	X =  321.485  mm,	Y =   -468.955  mm,	Z =   -267.000  mm,
	W =  90.000 deg,	P =   0.000 deg,	R =   90.000 deg
};
P[439]{
   GP1:
	UF : 0, UT : 6,		CONFIG : 'N U T, 0, 0, 0',
	X =  303.278  mm,	Y =   -479.431  mm,	Z =   -267.000  mm,
	W =  90.000 deg,	P =   0.000 deg,	R =   90.000 deg
};
P[440]{
   GP1:
	UF : 0, UT : 6,		CONFIG : 'N U T, 0, 0, 0',
	X =  248.887  mm,	Y =   -510.794  mm,	Z =   -267.000  mm,
	W =  90.000 deg,	P =   0.000 deg,	R =   90.000 deg
};
P[441]{
   GP1:
	UF : 0, UT : 6,		CONFIG : 'N U T, 0, 0, 0',
	X =  230.541  mm,	Y =   -521.505  mm,	Z =   -267.000  mm,
	W =  90.000 deg,	P =   0.000 deg,	R =   90.000 deg
};
P[442]{
   GP1:
	UF : 0, UT : 6,		CONFIG : 'N U T, 0, 0, 0',
	X =  194.065  mm,	Y =   -542.556  mm,	Z =   -267.000  mm,
	W =  90.000 deg,	P =   0.000 deg,	R =   90.000 deg
};
P[443]{
   GP1:
	UF : 0, UT : 6,		CONFIG : 'N U T, 0, 0, 0',
	X =  139.530  mm,	Y =   -573.935  mm,	Z =   -267.000  mm,
	W =  90.000 deg,	P =   0.000 deg,	R =   90.000 deg
};
P[444]{
   GP1:
	UF : 0, UT : 6,		CONFIG : 'N U T, 0, 0, 0',
	X =  121.558  mm,	Y =   -584.313  mm,	Z =   -267.000  mm,
	W =  90.000 deg,	P =   0.000 deg,	R =   90.000 deg
};
P[445]{
   GP1:
	UF : 0, UT : 6,		CONFIG : 'N U T, 0, 0, 0',
	X =  69.455  mm,	Y =   -614.511  mm,	Z =   -248.193  mm,
	W =  90.000 deg,	P =   0.000 deg,	R =   90.000 deg
};
P[446]{
   GP1:
	UF : 0, UT : 6,		CONFIG : 'N U T, 0, 0, 0',
	X =  73.807  mm,	Y =   -612.144  mm,	Z =   -261.927  mm,
	W =  90.000 deg,	P =   0.000 deg,	R =   90.000 deg
};
P[447]{
   GP1:
	UF : 0, UT : 6,		CONFIG : 'N U T, 0, 0, 0',
	X =  85.175  mm,	Y =   -605.574  mm,	Z =   -266.999  mm,
	W =  90.000 deg,	P =   0.000 deg,	R =   90.000 deg
};
P[448]{
   GP1:
	UF : 0, UT : 6,		CONFIG : 'N U T, 0, 0, 0',
	X =  103.342  mm,	Y =   -595.091  mm,	Z =   -267.000  mm,
	W =  90.000 deg,	P =   0.000 deg,	R =   90.000 deg
};
P[449]{
   GP1:
	UF : 0, UT : 6,		CONFIG : 'N U T, 0, 0, 0',
	X =  158.046  mm,	Y =   -563.598  mm,	Z =   -267.000  mm,
	W =  90.000 deg,	P =   0.000 deg,	R =   90.000 deg
};
P[450]{
   GP1:
	UF : 0, UT : 6,		CONFIG : 'N U T, 0, 0, 0',
	X =  176.088  mm,	Y =   -553.101  mm,	Z =   -267.000  mm,
	W =  90.000 deg,	P =   0.000 deg,	R =   90.000 deg
};
P[451]{
   GP1:
	UF : 0, UT : 6,		CONFIG : 'N U T, 0, 0, 0',
	X =  212.495  mm,	Y =   -531.950  mm,	Z =   -267.000  mm,
	W =  90.000 deg,	P =   0.000 deg,	R =   90.000 deg
};
P[452]{
   GP1:
	UF : 0, UT : 6,		CONFIG : 'N U T, 0, 0, 0',
	X =  266.860  mm,	Y =   -500.614  mm,	Z =   -267.000  mm,
	W =  90.000 deg,	P =   0.000 deg,	R =   90.000 deg
};
P[453]{
   GP1:
	UF : 0, UT : 6,		CONFIG : 'N U T, 0, 0, 0',
	X =  285.368  mm,	Y =   -490.006  mm,	Z =   -267.000  mm,
	W =  90.000 deg,	P =   0.000 deg,	R =   90.000 deg
};
P[454]{
   GP1:
	UF : 0, UT : 6,		CONFIG : 'N U T, 0, 0, 0',
	X =  339.837  mm,	Y =   -458.448  mm,	Z =   -267.000  mm,
	W =  90.000 deg,	P =   0.000 deg,	R =   90.000 deg
};
P[455]{
   GP1:
	UF : 0, UT : 6,		CONFIG : 'N U T, 0, 0, 0',
	X =  357.990  mm,	Y =   -448.207  mm,	Z =   -267.000  mm,
	W =  90.000 deg,	P =   0.000 deg,	R =   90.000 deg
};
P[456]{
   GP1:
	UF : 0, UT : 6,		CONFIG : 'N U T, 0, 0, 0',
	X =  376.120  mm,	Y =   -437.531  mm,	Z =   -267.000  mm,
	W =  90.000 deg,	P =   0.000 deg,	R =   90.000 deg
};
P[457]{
   GP1:
	UF : 0, UT : 6,		CONFIG : 'N U T, 0, 0, 0',
	X =  394.238  mm,	Y =   -427.152  mm,	Z =   -267.000  mm,
	W =  90.000 deg,	P =   0.000 deg,	R =   90.000 deg
};
P[458]{
   GP1:
	UF : 0, UT : 6,		CONFIG : 'N U T, 0, 0, 0',
	X =  412.785  mm,	Y =   -416.547  mm,	Z =   -267.000  mm,
	W =  90.000 deg,	P =   0.000 deg,	R =   90.000 deg
};
P[459]{
   GP1:
	UF : 0, UT : 6,		CONFIG : 'N U T, 0, 0, 0',
	X =  448.959  mm,	Y =   -395.706  mm,	Z =   -267.000  mm,
	W =  90.000 deg,	P =   0.000 deg,	R =   90.000 deg
};
P[460]{
   GP1:
	UF : 0, UT : 6,		CONFIG : 'N U T, 0, 0, 0',
	X =  485.175  mm,	Y =   -374.654  mm,	Z =   -267.000  mm,
	W =  90.000 deg,	P =   0.000 deg,	R =   90.000 deg
};
P[461]{
   GP1:
	UF : 0, UT : 6,		CONFIG : 'N U T, 0, 0, 0',
	X =  521.461  mm,	Y =   -353.543  mm,	Z =   -267.000  mm,
	W =  90.000 deg,	P =   0.000 deg,	R =   90.000 deg
};
P[462]{
   GP1:
	UF : 0, UT : 6,		CONFIG : 'N U T, 0, 0, 0',
	X =  581.548  mm,	Y =   -343.057  mm,	Z =   -248.136  mm,
	W =  90.000 deg,	P =   0.000 deg,	R =   90.000 deg
};
P[463]{
   GP1:
	UF : 0, UT : 6,		CONFIG : 'N U T, 0, 0, 0',
	X =  569.674  mm,	Y =   -349.887  mm,	Z =   -266.231  mm,
	W =  90.000 deg,	P =   0.000 deg,	R =   90.000 deg
};
P[464]{
   GP1:
	UF : 0, UT : 6,		CONFIG : 'N U T, 0, 0, 0',
	X =  495.732  mm,	Y =   -392.513  mm,	Z =   -267.000  mm,
	W =  90.000 deg,	P =   0.000 deg,	R =   90.000 deg
};
P[465]{
   GP1:
	UF : 0, UT : 6,		CONFIG : 'N U T, 0, 0, 0',
	X =  477.461  mm,	Y =   -403.017  mm,	Z =   -267.000  mm,
	W =  90.000 deg,	P =   0.000 deg,	R =   90.000 deg
};
P[466]{
   GP1:
	UF : 0, UT : 6,		CONFIG : 'N U T, 0, 0, 0',
	X =  441.221  mm,	Y =   -424.060  mm,	Z =   -267.000  mm,
	W =  90.000 deg,	P =   0.000 deg,	R =   90.000 deg
};
P[467]{
   GP1:
	UF : 0, UT : 6,		CONFIG : 'N U T, 0, 0, 0',
	X =  404.597  mm,	Y =   -445.232  mm,	Z =   -267.000  mm,
	W =  90.000 deg,	P =   0.000 deg,	R =   90.000 deg
};
P[468]{
   GP1:
	UF : 0, UT : 6,		CONFIG : 'N U T, 0, 0, 0',
	X =  386.626  mm,	Y =   -455.612  mm,	Z =   -267.000  mm,
	W =  90.000 deg,	P =   0.000 deg,	R =   90.000 deg
};
P[469]{
   GP1:
	UF : 0, UT : 6,		CONFIG : 'N U T, 0, 0, 0',
	X =  368.349  mm,	Y =   -466.118  mm,	Z =   -267.000  mm,
	W =  90.000 deg,	P =   0.000 deg,	R =   90.000 deg
};
P[470]{
   GP1:
	UF : 0, UT : 6,		CONFIG : 'N U T, 0, 0, 0',
	X =  350.098  mm,	Y =   -476.669  mm,	Z =   -267.000  mm,
	W =  90.000 deg,	P =   0.000 deg,	R =   90.000 deg
};
P[471]{
   GP1:
	UF : 0, UT : 6,		CONFIG : 'N U T, 0, 0, 0',
	X =  313.809  mm,	Y =   -497.611  mm,	Z =   -267.000  mm,
	W =  90.000 deg,	P =   0.000 deg,	R =   90.000 deg
};
P[472]{
   GP1:
	UF : 0, UT : 6,		CONFIG : 'N U T, 0, 0, 0',
	X =  259.253  mm,	Y =   -529.033  mm,	Z =   -267.000  mm,
	W =  90.000 deg,	P =   0.000 deg,	R =   90.000 deg
};
P[473]{
   GP1:
	UF : 0, UT : 6,		CONFIG : 'N U T, 0, 0, 0',
	X =  240.975  mm,	Y =   -539.441  mm,	Z =   -267.000  mm,
	W =  90.000 deg,	P =   0.000 deg,	R =   90.000 deg
};
P[474]{
   GP1:
	UF : 0, UT : 6,		CONFIG : 'N U T, 0, 0, 0',
	X =  186.337  mm,	Y =   -571.044  mm,	Z =   -267.000  mm,
	W =  90.000 deg,	P =   0.000 deg,	R =   90.000 deg
};
P[475]{
   GP1:
	UF : 0, UT : 6,		CONFIG : 'N U T, 0, 0, 0',
	X =  131.747  mm,	Y =   -602.648  mm,	Z =   -267.000  mm,
	W =  90.000 deg,	P =   0.000 deg,	R =   90.000 deg
};
P[476]{
   GP1:
	UF : 0, UT : 6,		CONFIG : 'N U T, 0, 0, 0',
	X =  113.540  mm,	Y =   -613.030  mm,	Z =   -267.000  mm,
	W =  90.000 deg,	P =   0.000 deg,	R =   90.000 deg
};
P[477]{
   GP1:
	UF : 0, UT : 6,		CONFIG : 'N U T, 0, 0, 0',
	X =  79.956  mm,	Y =   -632.694  mm,	Z =   -248.200  mm,
	W =  90.000 deg,	P =   0.000 deg,	R =   90.000 deg
};
P[478]{
   GP1:
	UF : 0, UT : 6,		CONFIG : 'N U T, 0, 0, 0',
	X =  84.360  mm,	Y =   -630.389  mm,	Z =   -261.973  mm,
	W =  90.000 deg,	P =   0.000 deg,	R =   90.000 deg
};
P[479]{
   GP1:
	UF : 0, UT : 6,		CONFIG : 'N U T, 0, 0, 0',
	X =  95.519  mm,	Y =   -623.823  mm,	Z =   -266.999  mm,
	W =  90.000 deg,	P =   0.000 deg,	R =   90.000 deg
};
P[480]{
   GP1:
	UF : 0, UT : 6,		CONFIG : 'N U T, 0, 0, 0',
	X =  150.126  mm,	Y =   -592.253  mm,	Z =   -267.000  mm,
	W =  90.000 deg,	P =   0.000 deg,	R =   90.000 deg
};
P[481]{
   GP1:
	UF : 0, UT : 6,		CONFIG : 'N U T, 0, 0, 0',
	X =  168.419  mm,	Y =   -581.719  mm,	Z =   -267.000  mm,
	W =  90.000 deg,	P =   0.000 deg,	R =   90.000 deg
};
P[482]{
   GP1:
	UF : 0, UT : 6,		CONFIG : 'N U T, 0, 0, 0',
	X =  204.831  mm,	Y =   -560.612  mm,	Z =   -267.000  mm,
	W =  90.000 deg,	P =   0.000 deg,	R =   90.000 deg
};
P[483]{
   GP1:
	UF : 0, UT : 6,		CONFIG : 'N U T, 0, 0, 0',
	X =  223.052  mm,	Y =   -550.261  mm,	Z =   -267.000  mm,
	W =  90.000 deg,	P =   0.000 deg,	R =   90.000 deg
};
P[484]{
   GP1:
	UF : 0, UT : 6,		CONFIG : 'N U T, 0, 0, 0',
	X =  277.625  mm,	Y =   -518.677  mm,	Z =   -267.000  mm,
	W =  90.000 deg,	P =   0.000 deg,	R =   90.000 deg
};
P[485]{
   GP1:
	UF : 0, UT : 6,		CONFIG : 'N U T, 0, 0, 0',
	X =  295.801  mm,	Y =   -508.256  mm,	Z =   -267.000  mm,
	W =  90.000 deg,	P =   0.000 deg,	R =   90.000 deg
};
P[486]{
   GP1:
	UF : 0, UT : 6,		CONFIG : 'N U T, 0, 0, 0',
	X =  332.180  mm,	Y =   -487.237  mm,	Z =   -267.000  mm,
	W =  90.000 deg,	P =   0.000 deg,	R =   90.000 deg
};
P[487]{
   GP1:
	UF : 0, UT : 6,		CONFIG : 'N U T, 0, 0, 0',
	X =  422.842  mm,	Y =   -434.745  mm,	Z =   -267.000  mm,
	W =  90.000 deg,	P =   0.000 deg,	R =   90.000 deg
};
P[488]{
   GP1:
	UF : 0, UT : 6,		CONFIG : 'N U T, 0, 0, 0',
	X =  459.065  mm,	Y =   -413.887  mm,	Z =   -267.000  mm,
	W =  90.000 deg,	P =   0.000 deg,	R =   90.000 deg
};
P[489]{
   GP1:
	UF : 0, UT : 6,		CONFIG : 'N U T, 0, 0, 0',
	X =  514.184  mm,	Y =   -382.024  mm,	Z =   -267.000  mm,
	W =  90.000 deg,	P =   0.000 deg,	R =   90.000 deg
};
P[490]{
   GP1:
	UF : 0, UT : 6,		CONFIG : 'N U T, 0, 0, 0',
	X =  532.228  mm,	Y =   -371.647  mm,	Z =   -267.000  mm,
	W =  90.000 deg,	P =   0.000 deg,	R =   90.000 deg
};
P[491]{
   GP1:
	UF : 0, UT : 6,		CONFIG : 'N U T, 0, 0, 0',
	X =  550.141  mm,	Y =   -361.240  mm,	Z =   -267.000  mm,
	W =  90.000 deg,	P =   0.000 deg,	R =   90.000 deg
};
P[492]{
   GP1:
	UF : 0, UT : 6,		CONFIG : 'N U T, 0, 0, 0',
	X =  578.422  mm,	Y =   -345.240  mm,	Z =   -258.781  mm,
	W =  90.000 deg,	P =   0.000 deg,	R =   90.000 deg
};
P[493]{
   GP1:
	UF : 0, UT : 6,		CONFIG : 'N U T, 0, 0, 0',
	X =  580.211  mm,	Y =   -368.067  mm,	Z =   -266.283  mm,
	W =  90.000 deg,	P =   0.000 deg,	R =   90.000 deg
};
P[494]{
   GP1:
	UF : 0, UT : 6,		CONFIG : 'N U T, 0, 0, 0',
	X =  560.695  mm,	Y =   -379.290  mm,	Z =   -267.000  mm,
	W =  90.000 deg,	P =   0.000 deg,	R =   90.000 deg
};
P[495]{
   GP1:
	UF : 0, UT : 6,		CONFIG : 'N U T, 0, 0, 0',
	X =  505.985  mm,	Y =   -410.945  mm,	Z =   -267.000  mm,
	W =  90.000 deg,	P =   0.000 deg,	R =   90.000 deg
};
P[496]{
   GP1:
	UF : 0, UT : 6,		CONFIG : 'N U T, 0, 0, 0',
	X =  469.806  mm,	Y =   -431.829  mm,	Z =   -267.000  mm,
	W =  90.000 deg,	P =   0.000 deg,	R =   90.000 deg
};
P[497]{
   GP1:
	UF : 0, UT : 6,		CONFIG : 'N U T, 0, 0, 0',
	X =  396.987  mm,	Y =   -473.854  mm,	Z =   -267.000  mm,
	W =  90.000 deg,	P =   0.000 deg,	R =   90.000 deg
};
P[498]{
   GP1:
	UF : 0, UT : 6,		CONFIG : 'N U T, 0, 0, 0',
	X =  360.530  mm,	Y =   -494.814  mm,	Z =   -267.000  mm,
	W =  90.000 deg,	P =   0.000 deg,	R =   90.000 deg
};
P[499]{
   GP1:
	UF : 0, UT : 6,		CONFIG : 'N U T, 0, 0, 0',
	X =  342.478  mm,	Y =   -505.311  mm,	Z =   -267.000  mm,
	W =  90.000 deg,	P =   0.000 deg,	R =   90.000 deg
};
P[500]{
   GP1:
	UF : 0, UT : 6,		CONFIG : 'N U T, 0, 0, 0',
	X =  324.052  mm,	Y =   -515.696  mm,	Z =   -267.000  mm,
	W =  90.000 deg,	P =   0.000 deg,	R =   90.000 deg
};
P[501]{
   GP1:
	UF : 0, UT : 6,		CONFIG : 'N U T, 0, 0, 0',
	X =  306.123  mm,	Y =   -526.319  mm,	Z =   -267.000  mm,
	W =  90.000 deg,	P =   0.000 deg,	R =   90.000 deg
};
P[502]{
   GP1:
	UF : 0, UT : 6,		CONFIG : 'N U T, 0, 0, 0',
	X =  287.949  mm,	Y =   -536.712  mm,	Z =   -267.000  mm,
	W =  90.000 deg,	P =   0.000 deg,	R =   90.000 deg
};
P[503]{
   GP1:
	UF : 0, UT : 6,		CONFIG : 'N U T, 0, 0, 0',
	X =  251.698  mm,	Y =   -557.782  mm,	Z =   -267.000  mm,
	W =  90.000 deg,	P =   0.000 deg,	R =   90.000 deg
};
P[504]{
   GP1:
	UF : 0, UT : 6,		CONFIG : 'N U T, 0, 0, 0',
	X =  215.213  mm,	Y =   -578.773  mm,	Z =   -267.000  mm,
	W =  90.000 deg,	P =   0.000 deg,	R =   90.000 deg
};
P[505]{
   GP1:
	UF : 0, UT : 6,		CONFIG : 'N U T, 0, 0, 0',
	X =  160.535  mm,	Y =   -610.339  mm,	Z =   -267.000  mm,
	W =  90.000 deg,	P =   0.000 deg,	R =   90.000 deg
};
P[506]{
   GP1:
	UF : 0, UT : 6,		CONFIG : 'N U T, 0, 0, 0',
	X =  142.213  mm,	Y =   -620.805  mm,	Z =   -267.000  mm,
	W =  90.000 deg,	P =   0.000 deg,	R =   90.000 deg
};
P[507]{
   GP1:
	UF : 0, UT : 6,		CONFIG : 'N U T, 0, 0, 0',
	X =  106.162  mm,	Y =   -641.800  mm,	Z =   -266.999  mm,
	W =  90.000 deg,	P =   0.000 deg,	R =   90.000 deg
};
P[508]{
   GP1:
	UF : 0, UT : 6,		CONFIG : 'N U T, 0, 0, 0',
	X =  94.773  mm,	Y =   -648.395  mm,	Z =   -262.002  mm,
	W =  90.000 deg,	P =   0.000 deg,	R =   90.000 deg
};
P[509]{
   GP1:
	UF : 0, UT : 6,		CONFIG : 'N U T, 0, 0, 0',
	X =  90.472  mm,	Y =   -650.908  mm,	Z =   -248.200  mm,
	W =  90.000 deg,	P =   0.000 deg,	R =   90.000 deg
};
P[510]{
   GP1:
	UF : 0, UT : 6,		CONFIG : 'N U T, 0, 0, 0',
	X =  124.271  mm,	Y =   -631.447  mm,	Z =   -267.000  mm,
	W =  90.000 deg,	P =   0.000 deg,	R =   90.000 deg
};
P[511]{
   GP1:
	UF : 0, UT : 6,		CONFIG : 'N U T, 0, 0, 0',
	X =  178.773  mm,	Y =   -600.003  mm,	Z =   -267.000  mm,
	W =  90.000 deg,	P =   0.000 deg,	R =   90.000 deg
};
P[512]{
   GP1:
	UF : 0, UT : 6,		CONFIG : 'N U T, 0, 0, 0',
	X =  196.986  mm,	Y =   -589.631  mm,	Z =   -267.000  mm,
	W =  90.000 deg,	P =   0.000 deg,	R =   90.000 deg
};
P[513]{
   GP1:
	UF : 0, UT : 6,		CONFIG : 'N U T, 0, 0, 0',
	X =  233.418  mm,	Y =   -568.352  mm,	Z =   -267.000  mm,
	W =  90.000 deg,	P =   0.000 deg,	R =   90.000 deg
};
P[514]{
   GP1:
	UF : 0, UT : 6,		CONFIG : 'N U T, 0, 0, 0',
	X =  269.919  mm,	Y =   -547.346  mm,	Z =   -267.000  mm,
	W =  90.000 deg,	P =   0.000 deg,	R =   90.000 deg
};
P[515]{
   GP1:
	UF : 0, UT : 6,		CONFIG : 'N U T, 0, 0, 0',
	X =  378.875  mm,	Y =   -484.547  mm,	Z =   -267.000  mm,
	W =  90.000 deg,	P =   0.000 deg,	R =   90.000 deg
};
P[516]{
   GP1:
	UF : 0, UT : 6,		CONFIG : 'N U T, 0, 0, 0',
	X =  415.424  mm,	Y =   -463.320  mm,	Z =   -267.000  mm,
	W =  90.000 deg,	P =   0.000 deg,	R =   90.000 deg
};
P[517]{
   GP1:
	UF : 0, UT : 6,		CONFIG : 'N U T, 0, 0, 0',
	X =  433.559  mm,	Y =   -452.991  mm,	Z =   -267.000  mm,
	W =  90.000 deg,	P =   0.000 deg,	R =   90.000 deg
};
P[518]{
   GP1:
	UF : 0, UT : 6,		CONFIG : 'N U T, 0, 0, 0',
	X =  451.784  mm,	Y =   -442.412  mm,	Z =   -267.000  mm,
	W =  90.000 deg,	P =   0.000 deg,	R =   90.000 deg
};
P[519]{
   GP1:
	UF : 0, UT : 6,		CONFIG : 'N U T, 0, 0, 0',
	X =  488.126  mm,	Y =   -421.292  mm,	Z =   -267.000  mm,
	W =  90.000 deg,	P =   0.000 deg,	R =   90.000 deg
};
P[520]{
   GP1:
	UF : 0, UT : 6,		CONFIG : 'N U T, 0, 0, 0',
	X =  524.439  mm,	Y =   -400.389  mm,	Z =   -267.000  mm,
	W =  90.000 deg,	P =   0.000 deg,	R =   90.000 deg
};
P[521]{
   GP1:
	UF : 0, UT : 6,		CONFIG : 'N U T, 0, 0, 0',
	X =  542.644  mm,	Y =   -390.001  mm,	Z =   -267.000  mm,
	W =  90.000 deg,	P =   0.000 deg,	R =   90.000 deg
};
P[522]{
   GP1:
	UF : 0, UT : 6,		CONFIG : 'N U T, 0, 0, 0',
	X =  588.832  mm,	Y =   -363.325  mm,	Z =   -258.859  mm,
	W =  90.000 deg,	P =   0.000 deg,	R =   90.000 deg
};
P[523]{
   GP1:
	UF : 0, UT : 6,		CONFIG : 'N U T, 0, 0, 0',
	X =  592.208  mm,	Y =   -361.394  mm,	Z =   -247.960  mm,
	W =  90.000 deg,	P =   0.000 deg,	R =   90.000 deg
};
P[524]{
   GP1:
	UF : 0, UT : 6,		CONFIG : 'N U T, 0, 0, 0',
	X =  602.472  mm,	Y =   -379.509  mm,	Z =   -248.435  mm,
	W =  90.000 deg,	P =   0.000 deg,	R =   90.000 deg
};
P[525]{
   GP1:
	UF : 0, UT : 6,		CONFIG : 'N U T, 0, 0, 0',
	X =  534.847  mm,	Y =   -418.347  mm,	Z =   -267.000  mm,
	W =  90.000 deg,	P =   0.000 deg,	R =   90.000 deg
};
P[526]{
   GP1:
	UF : 0, UT : 6,		CONFIG : 'N U T, 0, 0, 0',
	X =  498.274  mm,	Y =   -439.482  mm,	Z =   -267.000  mm,
	W =  90.000 deg,	P =   0.000 deg,	R =   90.000 deg
};
P[527]{
   GP1:
	UF : 0, UT : 6,		CONFIG : 'N U T, 0, 0, 0',
	X =  407.652  mm,	Y =   -491.986  mm,	Z =   -267.000  mm,
	W =  90.000 deg,	P =   0.000 deg,	R =   90.000 deg
};
P[528]{
   GP1:
	UF : 0, UT : 6,		CONFIG : 'N U T, 0, 0, 0',
	X =  389.393  mm,	Y =   -502.496  mm,	Z =   -267.000  mm,
	W =  90.000 deg,	P =   0.000 deg,	R =   90.000 deg
};
P[529]{
   GP1:
	UF : 0, UT : 6,		CONFIG : 'N U T, 0, 0, 0',
	X =  352.833  mm,	Y =   -523.469  mm,	Z =   -267.000  mm,
	W =  90.000 deg,	P =   0.000 deg,	R =   90.000 deg
};
P[530]{
   GP1:
	UF : 0, UT : 6,		CONFIG : 'N U T, 0, 0, 0',
	X =  316.604  mm,	Y =   -544.429  mm,	Z =   -267.000  mm,
	W =  90.000 deg,	P =   0.000 deg,	R =   90.000 deg
};
P[531]{
   GP1:
	UF : 0, UT : 6,		CONFIG : 'N U T, 0, 0, 0',
	X =  280.341  mm,	Y =   -565.474  mm,	Z =   -267.000  mm,
	W =  90.000 deg,	P =   0.000 deg,	R =   90.000 deg
};
P[532]{
   GP1:
	UF : 0, UT : 6,		CONFIG : 'N U T, 0, 0, 0',
	X =  243.658  mm,	Y =   -586.484  mm,	Z =   -267.000  mm,
	W =  90.000 deg,	P =   0.000 deg,	R =   90.000 deg
};
P[533]{
   GP1:
	UF : 0, UT : 6,		CONFIG : 'N U T, 0, 0, 0',
	X =  225.600  mm,	Y =   -596.805  mm,	Z =   -267.000  mm,
	W =  90.000 deg,	P =   0.000 deg,	R =   90.000 deg
};
P[534]{
   GP1:
	UF : 0, UT : 6,		CONFIG : 'N U T, 0, 0, 0',
	X =  207.565  mm,	Y =   -607.525  mm,	Z =   -267.000  mm,
	W =  90.000 deg,	P =   0.000 deg,	R =   90.000 deg
};
P[535]{
   GP1:
	UF : 0, UT : 6,		CONFIG : 'N U T, 0, 0, 0',
	X =  134.641  mm,	Y =   -649.517  mm,	Z =   -267.000  mm,
	W =  90.000 deg,	P =   0.000 deg,	R =   90.000 deg
};
P[536]{
   GP1:
	UF : 0, UT : 6,		CONFIG : 'N U T, 0, 0, 0',
	X =  116.667  mm,	Y =   -659.834  mm,	Z =   -266.999  mm,
	W =  90.000 deg,	P =   0.000 deg,	R =   90.000 deg
};
P[537]{
   GP1:
	UF : 0, UT : 6,		CONFIG : 'N U T, 0, 0, 0',
	X =  100.943  mm,	Y =   -669.018  mm,	Z =   -248.233  mm,
	W =  90.000 deg,	P =   0.000 deg,	R =   90.000 deg
};
P[538]{
   GP1:
	UF : 0, UT : 6,		CONFIG : 'N U T, 0, 0, 0',
	X =  105.313  mm,	Y =   -666.641  mm,	Z =   -261.991  mm,
	W =  90.000 deg,	P =   0.000 deg,	R =   90.000 deg
};
P[539]{
   GP1:
	UF : 0, UT : 6,		CONFIG : 'N U T, 0, 0, 0',
	X =  152.979  mm,	Y =   -639.046  mm,	Z =   -267.000  mm,
	W =  90.000 deg,	P =   0.000 deg,	R =   90.000 deg
};
P[540]{
   GP1:
	UF : 0, UT : 6,		CONFIG : 'N U T, 0, 0, 0',
	X =  171.400  mm,	Y =   -628.527  mm,	Z =   -267.000  mm,
	W =  90.000 deg,	P =   0.000 deg,	R =   90.000 deg
};
P[541]{
   GP1:
	UF : 0, UT : 6,		CONFIG : 'N U T, 0, 0, 0',
	X =  189.254  mm,	Y =   -618.287  mm,	Z =   -267.000  mm,
	W =  90.000 deg,	P =   0.000 deg,	R =   90.000 deg
};
P[542]{
   GP1:
	UF : 0, UT : 6,		CONFIG : 'N U T, 0, 0, 0',
	X =  261.985  mm,	Y =   -576.181  mm,	Z =   -267.000  mm,
	W =  90.000 deg,	P =   0.000 deg,	R =   90.000 deg
};
P[543]{
   GP1:
	UF : 0, UT : 6,		CONFIG : 'N U T, 0, 0, 0',
	X =  298.625  mm,	Y =   -555.072  mm,	Z =   -267.000  mm,
	W =  90.000 deg,	P =   0.000 deg,	R =   90.000 deg
};
P[544]{
   GP1:
	UF : 0, UT : 6,		CONFIG : 'N U T, 0, 0, 0',
	X =  334.764  mm,	Y =   -534.219  mm,	Z =   -267.000  mm,
	W =  90.000 deg,	P =   0.000 deg,	R =   90.000 deg
};
P[545]{
   GP1:
	UF : 0, UT : 6,		CONFIG : 'N U T, 0, 0, 0',
	X =  371.261  mm,	Y =   -513.223  mm,	Z =   -267.000  mm,
	W =  90.000 deg,	P =   0.000 deg,	R =   90.000 deg
};
P[546]{
   GP1:
	UF : 0, UT : 6,		CONFIG : 'N U T, 0, 0, 0',
	X =  425.865  mm,	Y =   -481.595  mm,	Z =   -267.000  mm,
	W =  90.000 deg,	P =   0.000 deg,	R =   90.000 deg
};
P[547]{
   GP1:
	UF : 0, UT : 6,		CONFIG : 'N U T, 0, 0, 0',
	X =  443.907  mm,	Y =   -471.071  mm,	Z =   -267.000  mm,
	W =  90.000 deg,	P =   0.000 deg,	R =   90.000 deg
};
P[548]{
   GP1:
	UF : 0, UT : 6,		CONFIG : 'N U T, 0, 0, 0',
	X =  462.413  mm,	Y =   -460.660  mm,	Z =   -267.000  mm,
	W =  90.000 deg,	P =   0.000 deg,	R =   90.000 deg
};
P[549]{
   GP1:
	UF : 0, UT : 6,		CONFIG : 'N U T, 0, 0, 0',
	X =  480.379  mm,	Y =   -450.110  mm,	Z =   -267.000  mm,
	W =  90.000 deg,	P =   0.000 deg,	R =   90.000 deg
};
P[550]{
   GP1:
	UF : 0, UT : 6,		CONFIG : 'N U T, 0, 0, 0',
	X =  516.735  mm,	Y =   -429.024  mm,	Z =   -267.000  mm,
	W =  90.000 deg,	P =   0.000 deg,	R =   90.000 deg
};
P[551]{
   GP1:
	UF : 0, UT : 6,		CONFIG : 'N U T, 0, 0, 0',
	X =  553.156  mm,	Y =   -408.024  mm,	Z =   -267.000  mm,
	W =  90.000 deg,	P =   0.000 deg,	R =   90.000 deg
};
P[552]{
   GP1:
	UF : 0, UT : 6,		CONFIG : 'N U T, 0, 0, 0',
	X =  571.259  mm,	Y =   -397.553  mm,	Z =   -267.000  mm,
	W =  90.000 deg,	P =   0.000 deg,	R =   90.000 deg
};
P[553]{
   GP1:
	UF : 0, UT : 6,		CONFIG : 'N U T, 0, 0, 0',
	X =  590.661  mm,	Y =   -386.345  mm,	Z =   -266.291  mm,
	W =  90.000 deg,	P =   0.000 deg,	R =   90.000 deg
};
P[554]{
   GP1:
	UF : 0, UT : 6,		CONFIG : 'N U T, 0, 0, 0',
	X =  599.439  mm,	Y =   -381.688  mm,	Z =   -258.848  mm,
	W =  90.000 deg,	P =   0.000 deg,	R =   90.000 deg
};
P[555]{
   GP1:
	UF : 0, UT : 6,		CONFIG : 'N U T, 0, 0, 0',
	X =  613.031  mm,	Y =   -397.646  mm,	Z =   -248.218  mm,
	W =  90.000 deg,	P =   0.000 deg,	R =   90.000 deg
};
P[556]{
   GP1:
	UF : 0, UT : 6,		CONFIG : 'N U T, 0, 0, 0',
	X =  609.662  mm,	Y =   -399.413  mm,	Z =   -258.820  mm,
	W =  90.000 deg,	P =   0.000 deg,	R =   90.000 deg
};
P[557]{
   GP1:
	UF : 0, UT : 6,		CONFIG : 'N U T, 0, 0, 0',
	X =  601.279  mm,	Y =   -404.407  mm,	Z =   -266.188  mm,
	W =  90.000 deg,	P =   0.000 deg,	R =   90.000 deg
};
P[558]{
   GP1:
	UF : 0, UT : 6,		CONFIG : 'N U T, 0, 0, 0',
	X =  563.475  mm,	Y =   -426.232  mm,	Z =   -267.000  mm,
	W =  90.000 deg,	P =   0.000 deg,	R =   90.000 deg
};
P[559]{
   GP1:
	UF : 0, UT : 6,		CONFIG : 'N U T, 0, 0, 0',
	X =  545.385  mm,	Y =   -436.480  mm,	Z =   -267.000  mm,
	W =  90.000 deg,	P =   0.000 deg,	R =   90.000 deg
};
P[560]{
   GP1:
	UF : 0, UT : 6,		CONFIG : 'N U T, 0, 0, 0',
	X =  527.094  mm,	Y =   -447.219  mm,	Z =   -267.000  mm,
	W =  90.000 deg,	P =   0.000 deg,	R =   90.000 deg
};
P[561]{
   GP1:
	UF : 0, UT : 6,		CONFIG : 'N U T, 0, 0, 0',
	X =  490.749  mm,	Y =   -468.240  mm,	Z =   -267.000  mm,
	W =  90.000 deg,	P =   0.000 deg,	R =   90.000 deg
};
P[562]{
   GP1:
	UF : 0, UT : 6,		CONFIG : 'N U T, 0, 0, 0',
	X =  472.511  mm,	Y =   -478.629  mm,	Z =   -267.000  mm,
	W =  90.000 deg,	P =   0.000 deg,	R =   90.000 deg
};
P[563]{
   GP1:
	UF : 0, UT : 6,		CONFIG : 'N U T, 0, 0, 0',
	X =  436.400  mm,	Y =   -499.595  mm,	Z =   -267.000  mm,
	W =  90.000 deg,	P =   0.000 deg,	R =   90.000 deg
};
P[564]{
   GP1:
	UF : 0, UT : 6,		CONFIG : 'N U T, 0, 0, 0',
	X =  417.894  mm,	Y =   -509.996  mm,	Z =   -267.000  mm,
	W =  90.000 deg,	P =   0.000 deg,	R =   90.000 deg
};
P[565]{
   GP1:
	UF : 0, UT : 6,		CONFIG : 'N U T, 0, 0, 0',
	X =  400.063  mm,	Y =   -520.609  mm,	Z =   -267.000  mm,
	W =  90.000 deg,	P =   0.000 deg,	R =   90.000 deg
};
P[566]{
   GP1:
	UF : 0, UT : 6,		CONFIG : 'N U T, 0, 0, 0',
	X =  381.734  mm,	Y =   -531.150  mm,	Z =   -267.000  mm,
	W =  90.000 deg,	P =   0.000 deg,	R =   90.000 deg
};
P[567]{
   GP1:
	UF : 0, UT : 6,		CONFIG : 'N U T, 0, 0, 0',
	X =  345.355  mm,	Y =   -552.038  mm,	Z =   -267.000  mm,
	W =  90.000 deg,	P =   0.000 deg,	R =   90.000 deg
};
P[568]{
   GP1:
	UF : 0, UT : 6,		CONFIG : 'N U T, 0, 0, 0',
	X =  327.064  mm,	Y =   -562.724  mm,	Z =   -267.000  mm,
	W =  90.000 deg,	P =   0.000 deg,	R =   90.000 deg
};
P[569]{
   GP1:
	UF : 0, UT : 6,		CONFIG : 'N U T, 0, 0, 0',
	X =  309.028  mm,	Y =   -573.020  mm,	Z =   -267.000  mm,
	W =  90.000 deg,	P =   0.000 deg,	R =   90.000 deg
};
P[570]{
   GP1:
	UF : 0, UT : 6,		CONFIG : 'N U T, 0, 0, 0',
	X =  290.722  mm,	Y =   -583.743  mm,	Z =   -267.000  mm,
	W =  90.000 deg,	P =   0.000 deg,	R =   90.000 deg
};
P[571]{
   GP1:
	UF : 0, UT : 6,		CONFIG : 'N U T, 0, 0, 0',
	X =  218.035  mm,	Y =   -625.659  mm,	Z =   -267.000  mm,
	W =  90.000 deg,	P =   0.000 deg,	R =   90.000 deg
};
P[572]{
   GP1:
	UF : 0, UT : 6,		CONFIG : 'N U T, 0, 0, 0',
	X =  181.771  mm,	Y =   -646.647  mm,	Z =   -267.000  mm,
	W =  90.000 deg,	P =   0.000 deg,	R =   90.000 deg
};
P[573]{
   GP1:
	UF : 0, UT : 6,		CONFIG : 'N U T, 0, 0, 0',
	X =  163.332  mm,	Y =   -657.099  mm,	Z =   -267.000  mm,
	W =  90.000 deg,	P =   0.000 deg,	R =   90.000 deg
};
P[574]{
   GP1:
	UF : 0, UT : 6,		CONFIG : 'N U T, 0, 0, 0',
	X =  115.766  mm,	Y =   -684.709  mm,	Z =   -261.928  mm,
	W =  90.000 deg,	P =   0.000 deg,	R =   90.000 deg
};
P[575]{
   GP1:
	UF : 0, UT : 6,		CONFIG : 'N U T, 0, 0, 0',
	X =  111.446  mm,	Y =   -687.231  mm,	Z =   -248.194  mm,
	W =  90.000 deg,	P =   0.000 deg,	R =   90.000 deg
};
P[576]{
   GP1:
	UF : 0, UT : 6,		CONFIG : 'N U T, 0, 0, 0',
	X =  127.130  mm,	Y =   -678.303  mm,	Z =   -266.997  mm,
	W =  90.000 deg,	P =   0.000 deg,	R =   90.000 deg
};
P[577]{
   GP1:
	UF : 0, UT : 6,		CONFIG : 'N U T, 0, 0, 0',
	X =  145.400  mm,	Y =   -667.924  mm,	Z =   -267.000  mm,
	W =  90.000 deg,	P =   0.000 deg,	R =   90.000 deg
};
P[578]{
   GP1:
	UF : 0, UT : 6,		CONFIG : 'N U T, 0, 0, 0',
	X =  200.058  mm,	Y =   -636.256  mm,	Z =   -267.000  mm,
	W =  90.000 deg,	P =   0.000 deg,	R =   90.000 deg
};
P[579]{
   GP1:
	UF : 0, UT : 6,		CONFIG : 'N U T, 0, 0, 0',
	X =  236.169  mm,	Y =   -615.336  mm,	Z =   -267.000  mm,
	W =  90.000 deg,	P =   0.000 deg,	R =   90.000 deg
};
P[580]{
   GP1:
	UF : 0, UT : 6,		CONFIG : 'N U T, 0, 0, 0',
	X =  254.482  mm,	Y =   -604.846  mm,	Z =   -267.000  mm,
	W =  90.000 deg,	P =   0.000 deg,	R =   90.000 deg
};
P[581]{
   GP1:
	UF : 0, UT : 6,		CONFIG : 'N U T, 0, 0, 0',
	X =  272.771  mm,	Y =   -594.246  mm,	Z =   -267.000  mm,
	W =  90.000 deg,	P =   0.000 deg,	R =   90.000 deg
};
P[582]{
   GP1:
	UF : 0, UT : 6,		CONFIG : 'N U T, 0, 0, 0',
	X =  363.545  mm,	Y =   -541.924  mm,	Z =   -267.000  mm,
	W =  90.000 deg,	P =   0.000 deg,	R =   90.000 deg
};
P[583]{
   GP1:
	UF : 0, UT : 6,		CONFIG : 'N U T, 0, 0, 0',
	X =  454.522  mm,	Y =   -489.201  mm,	Z =   -267.000  mm,
	W =  90.000 deg,	P =   0.000 deg,	R =   90.000 deg
};
P[584]{
   GP1:
	UF : 0, UT : 6,		CONFIG : 'N U T, 0, 0, 0',
	X =  508.992  mm,	Y =   -457.956  mm,	Z =   -267.000  mm,
	W =  90.000 deg,	P =   0.000 deg,	R =   90.000 deg
};
P[585]{
   GP1:
	UF : 0, UT : 6,		CONFIG : 'N U T, 0, 0, 0',
	X =  582.042  mm,	Y =   -415.798  mm,	Z =   -267.000  mm,
	W =  90.000 deg,	P =   0.000 deg,	R =   90.000 deg
};
P[586]{
   GP1:
	UF : 0, UT : 6,		CONFIG : 'N U T, 0, 0, 0',
	X =  615.515  mm,	Y =   -409.900  mm,	Z =   -257.490  mm,
	W =  90.000 deg,	P =   0.000 deg,	R =   90.000 deg
};
P[587]{
   GP1:
	UF : 0, UT : 6,		CONFIG : 'N U T, 0, 0, 0',
	X =  123.196  mm,	Y =   -695.998  mm,	Z =   -259.674  mm,
	W =  90.000 deg,	P =   0.000 deg,	R =   90.000 deg
};
P[588]{
   GP1:
	UF : 0, UT : 6,		CONFIG : 'N U T, 0, 0, 0',
	X =  620.538  mm,	Y =   -412.751  mm,	Z =   -246.668  mm,
	W =  90.000 deg,	P =   0.000 deg,	R =   90.000 deg
};
P[589]{
   GP1:
	UF : 0, UT : 6,		CONFIG : 'N U T, 0, 0, 0',
	X =  608.041  mm,	Y =   -419.950  mm,	Z =   -263.147  mm,
	W =  90.000 deg,	P =   0.000 deg,	R =   90.000 deg
};
P[590]{
   GP1:
	UF : 0, UT : 6,		CONFIG : 'N U T, 0, 0, 0',
	X =  135.813  mm,	Y =   -693.181  mm,	Z =   -263.514  mm,
	W =  90.000 deg,	P =   0.000 deg,	R =   90.000 deg
};
P[591]{
   GP1:
	UF : 0, UT : 6,		CONFIG : 'N U T, 0, 0, 0',
	X =  154.251  mm,	Y =   -683.087  mm,	Z =   -263.903  mm,
	W =  90.000 deg,	P =   0.000 deg,	R =   90.000 deg
};
P[592]{
   GP1:
	UF : 0, UT : 6,		CONFIG : 'N U T, 0, 0, 0',
	X =  172.187  mm,	Y =   -672.838  mm,	Z =   -263.833  mm,
	W =  90.000 deg,	P =   0.000 deg,	R =   90.000 deg
};
P[593]{
   GP1:
	UF : 0, UT : 6,		CONFIG : 'N U T, 0, 0, 0',
	X =  190.582  mm,	Y =   -662.204  mm,	Z =   -263.818  mm,
	W =  90.000 deg,	P =   0.000 deg,	R =   90.000 deg
};
P[594]{
   GP1:
	UF : 0, UT : 6,		CONFIG : 'N U T, 0, 0, 0',
	X =  208.704  mm,	Y =   -651.654  mm,	Z =   -263.960  mm,
	W =  90.000 deg,	P =   0.000 deg,	R =   90.000 deg
};
P[595]{
   GP1:
	UF : 0, UT : 6,		CONFIG : 'N U T, 0, 0, 0',
	X =  226.972  mm,	Y =   -641.071  mm,	Z =   -263.921  mm,
	W =  90.000 deg,	P =   0.000 deg,	R =   90.000 deg
};
P[596]{
   GP1:
	UF : 0, UT : 6,		CONFIG : 'N U T, 0, 0, 0',
	X =  245.153  mm,	Y =   -630.600  mm,	Z =   -263.916  mm,
	W =  90.000 deg,	P =   0.000 deg,	R =   90.000 deg
};
P[597]{
   GP1:
	UF : 0, UT : 6,		CONFIG : 'N U T, 0, 0, 0',
	X =  263.255  mm,	Y =   -620.208  mm,	Z =   -263.839  mm,
	W =  90.000 deg,	P =   0.000 deg,	R =   90.000 deg
};
P[598]{
   GP1:
	UF : 0, UT : 6,		CONFIG : 'N U T, 0, 0, 0',
	X =  281.558  mm,	Y =   -609.622  mm,	Z =   -263.888  mm,
	W =  90.000 deg,	P =   0.000 deg,	R =   90.000 deg
};
P[599]{
   GP1:
	UF : 0, UT : 6,		CONFIG : 'N U T, 0, 0, 0',
	X =  299.655  mm,	Y =   -599.142  mm,	Z =   -263.881  mm,
	W =  90.000 deg,	P =   0.000 deg,	R =   90.000 deg
};
P[600]{
   GP1:
	UF : 0, UT : 6,		CONFIG : 'N U T, 0, 0, 0',
	X =  318.008  mm,	Y =   -588.573  mm,	Z =   -263.877  mm,
	W =  90.000 deg,	P =   0.000 deg,	R =   90.000 deg
};
P[601]{
   GP1:
	UF : 0, UT : 6,		CONFIG : 'N U T, 0, 0, 0',
	X =  335.973  mm,	Y =   -578.161  mm,	Z =   -263.902  mm,
	W =  90.000 deg,	P =   0.000 deg,	R =   90.000 deg
};
P[602]{
   GP1:
	UF : 0, UT : 6,		CONFIG : 'N U T, 0, 0, 0',
	X =  354.125  mm,	Y =   -567.711  mm,	Z =   -263.979  mm,
	W =  90.000 deg,	P =   0.000 deg,	R =   90.000 deg
};
P[603]{
   GP1:
	UF : 0, UT : 6,		CONFIG : 'N U T, 0, 0, 0',
	X =  372.539  mm,	Y =   -557.105  mm,	Z =   -263.848  mm,
	W =  90.000 deg,	P =   0.000 deg,	R =   90.000 deg
};
P[604]{
   GP1:
	UF : 0, UT : 6,		CONFIG : 'N U T, 0, 0, 0',
	X =  390.681  mm,	Y =   -546.605  mm,	Z =   -263.943  mm,
	W =  90.000 deg,	P =   0.000 deg,	R =   90.000 deg
};
P[605]{
   GP1:
	UF : 0, UT : 6,		CONFIG : 'N U T, 0, 0, 0',
	X =  408.686  mm,	Y =   -536.167  mm,	Z =   -263.883  mm,
	W =  90.000 deg,	P =   0.000 deg,	R =   90.000 deg
};
P[606]{
   GP1:
	UF : 0, UT : 6,		CONFIG : 'N U T, 0, 0, 0',
	X =  427.152  mm,	Y =   -525.556  mm,	Z =   -263.874  mm,
	W =  90.000 deg,	P =   0.000 deg,	R =   90.000 deg
};
P[607]{
   GP1:
	UF : 0, UT : 6,		CONFIG : 'N U T, 0, 0, 0',
	X =  445.340  mm,	Y =   -514.856  mm,	Z =   -264.027  mm,
	W =  90.000 deg,	P =   0.000 deg,	R =   90.000 deg
};
P[608]{
   GP1:
	UF : 0, UT : 6,		CONFIG : 'N U T, 0, 0, 0',
	X =  463.420  mm,	Y =   -504.764  mm,	Z =   -263.715  mm,
	W =  90.000 deg,	P =   0.000 deg,	R =   90.000 deg
};
P[609]{
   GP1:
	UF : 0, UT : 6,		CONFIG : 'N U T, 0, 0, 0',
	X =  481.657  mm,	Y =   -494.091  mm,	Z =   -263.787  mm,
	W =  90.000 deg,	P =   0.000 deg,	R =   90.000 deg
};
P[610]{
   GP1:
	UF : 0, UT : 6,		CONFIG : 'N U T, 0, 0, 0',
	X =  499.751  mm,	Y =   -483.759  mm,	Z =   -263.805  mm,
	W =  90.000 deg,	P =   0.000 deg,	R =   90.000 deg
};
P[611]{
   GP1:
	UF : 0, UT : 6,		CONFIG : 'N U T, 0, 0, 0',
	X =  518.153  mm,	Y =   -472.991  mm,	Z =   -263.913  mm,
	W =  90.000 deg,	P =   0.000 deg,	R =   90.000 deg
};
P[612]{
   GP1:
	UF : 0, UT : 6,		CONFIG : 'N U T, 0, 0, 0',
	X =  536.095  mm,	Y =   -462.579  mm,	Z =   -263.946  mm,
	W =  90.000 deg,	P =   0.000 deg,	R =   90.000 deg
};
P[613]{
   GP1:
	UF : 0, UT : 6,		CONFIG : 'N U T, 0, 0, 0',
	X =  554.182  mm,	Y =   -452.214  mm,	Z =   -263.790  mm,
	W =  90.000 deg,	P =   0.000 deg,	R =   90.000 deg
};
P[614]{
   GP1:
	UF : 0, UT : 6,		CONFIG : 'N U T, 0, 0, 0',
	X =  572.413  mm,	Y =   -441.810  mm,	Z =   -263.768  mm,
	W =  90.000 deg,	P =   0.000 deg,	R =   90.000 deg
};
P[615]{
   GP1:
	UF : 0, UT : 6,		CONFIG : 'N U T, 0, 0, 0',
	X =  590.873  mm,	Y =   -431.178  mm,	Z =   -263.744  mm,
	W =  90.000 deg,	P =   0.000 deg,	R =   90.000 deg
};
P[616]{
   GP1:
	UF : 0, UT : 6,		CONFIG : 'N U T, 0, 0, 0',
	X =  122.498  mm,	Y =   -701.908  mm,	Z =   -247.035  mm,
	W =  90.000 deg,	P =   0.000 deg,	R =   90.000 deg
};
P[617]{
   GP1:
	UF : 0, UT : 6,		CONFIG : 'N U T, 0, 0, 0',
	X =  139.304  mm,	Y =   -699.867  mm,	Z =   -248.273  mm,
	W =  90.000 deg,	P =   0.000 deg,	R =   90.000 deg
};
P[618]{
   GP1:
	UF : 0, UT : 6,		CONFIG : 'N U T, 0, 0, 0',
	X =  612.672  mm,	Y =   -425.956  mm,	Z =   -248.324  mm,
	W =  90.000 deg,	P =   0.000 deg,	R =   90.000 deg
};
P[619]{
   GP1:
	UF : 0, UT : 6,		CONFIG : 'N U T, 0, 0, 0',
	X =  594.237  mm,	Y =   -437.521  mm,	Z =   -248.124  mm,
	W =  90.000 deg,	P =   0.000 deg,	R =   90.000 deg
};
P[620]{
   GP1:
	UF : 0, UT : 6,		CONFIG : 'N U T, 0, 0, 0',
	X =  575.935  mm,	Y =   -448.000  mm,	Z =   -248.339  mm,
	W =  90.000 deg,	P =   0.000 deg,	R =   90.000 deg
};
P[621]{
   GP1:
	UF : 0, UT : 6,		CONFIG : 'N U T, 0, 0, 0',
	X =  557.988  mm,	Y =   -458.418  mm,	Z =   -248.204  mm,
	W =  90.000 deg,	P =   0.000 deg,	R =   90.000 deg
};
P[622]{
   GP1:
	UF : 0, UT : 6,		CONFIG : 'N U T, 0, 0, 0',
	X =  539.693  mm,	Y =   -469.028  mm,	Z =   -248.092  mm,
	W =  90.000 deg,	P =   0.000 deg,	R =   90.000 deg
};
P[623]{
   GP1:
	UF : 0, UT : 6,		CONFIG : 'N U T, 0, 0, 0',
	X =  521.416  mm,	Y =   -479.506  mm,	Z =   -248.272  mm,
	W =  90.000 deg,	P =   0.000 deg,	R =   90.000 deg
};
P[624]{
   GP1:
	UF : 0, UT : 6,		CONFIG : 'N U T, 0, 0, 0',
	X =  503.337  mm,	Y =   -489.937  mm,	Z =   -248.292  mm,
	W =  90.000 deg,	P =   0.000 deg,	R =   90.000 deg
};
P[625]{
   GP1:
	UF : 0, UT : 6,		CONFIG : 'N U T, 0, 0, 0',
	X =  485.444  mm,	Y =   -500.274  mm,	Z =   -248.278  mm,
	W =  90.000 deg,	P =   0.000 deg,	R =   90.000 deg
};
P[626]{
   GP1:
	UF : 0, UT : 6,		CONFIG : 'N U T, 0, 0, 0',
	X =  466.882  mm,	Y =   -510.956  mm,	Z =   -248.362  mm,
	W =  90.000 deg,	P =   0.000 deg,	R =   90.000 deg
};
P[627]{
   GP1:
	UF : 0, UT : 6,		CONFIG : 'N U T, 0, 0, 0',
	X =  448.850  mm,	Y =   -521.483  mm,	Z =   -248.083  mm,
	W =  90.000 deg,	P =   0.000 deg,	R =   90.000 deg
};
P[628]{
   GP1:
	UF : 0, UT : 6,		CONFIG : 'N U T, 0, 0, 0',
	X =  430.684  mm,	Y =   -531.923  mm,	Z =   -248.203  mm,
	W =  90.000 deg,	P =   0.000 deg,	R =   90.000 deg
};
P[629]{
   GP1:
	UF : 0, UT : 6,		CONFIG : 'N U T, 0, 0, 0',
	X =  412.531  mm,	Y =   -542.478  mm,	Z =   -248.024  mm,
	W =  90.000 deg,	P =   0.000 deg,	R =   90.000 deg
};
P[630]{
   GP1:
	UF : 0, UT : 6,		CONFIG : 'N U T, 0, 0, 0',
	X =  394.227  mm,	Y =   -552.947  mm,	Z =   -248.266  mm,
	W =  90.000 deg,	P =   0.000 deg,	R =   90.000 deg
};
P[631]{
   GP1:
	UF : 0, UT : 6,		CONFIG : 'N U T, 0, 0, 0',
	X =  376.065  mm,	Y =   -563.401  mm,	Z =   -248.344  mm,
	W =  90.000 deg,	P =   0.000 deg,	R =   90.000 deg
};
P[632]{
   GP1:
	UF : 0, UT : 6,		CONFIG : 'N U T, 0, 0, 0',
	X =  358.095  mm,	Y =   -573.896  mm,	Z =   -248.054  mm,
	W =  90.000 deg,	P =   0.000 deg,	R =   90.000 deg
};
P[633]{
   GP1:
	UF : 0, UT : 6,		CONFIG : 'N U T, 0, 0, 0',
	X =  339.863  mm,	Y =   -584.389  mm,	Z =   -248.137  mm,
	W =  90.000 deg,	P =   0.000 deg,	R =   90.000 deg
};
P[634]{
   GP1:
	UF : 0, UT : 6,		CONFIG : 'N U T, 0, 0, 0',
	X =  321.342  mm,	Y =   -595.078  mm,	Z =   -248.149  mm,
	W =  90.000 deg,	P =   0.000 deg,	R =   90.000 deg
};
P[635]{
   GP1:
	UF : 0, UT : 6,		CONFIG : 'N U T, 0, 0, 0',
	X =  303.180  mm,	Y =   -605.521  mm,	Z =   -248.253  mm,
	W =  90.000 deg,	P =   0.000 deg,	R =   90.000 deg
};
P[636]{
   GP1:
	UF : 0, UT : 6,		CONFIG : 'N U T, 0, 0, 0',
	X =  285.205  mm,	Y =   -615.969  mm,	Z =   -248.086  mm,
	W =  90.000 deg,	P =   0.000 deg,	R =   90.000 deg
};
P[637]{
   GP1:
	UF : 0, UT : 6,		CONFIG : 'N U T, 0, 0, 0',
	X =  266.932  mm,	Y =   -626.489  mm,	Z =   -248.162  mm,
	W =  90.000 deg,	P =   0.000 deg,	R =   90.000 deg
};
P[638]{
   GP1:
	UF : 0, UT : 6,		CONFIG : 'N U T, 0, 0, 0',
	X =  248.685  mm,	Y =   -637.035  mm,	Z =   -248.135  mm,
	W =  90.000 deg,	P =   0.000 deg,	R =   90.000 deg
};
P[639]{
   GP1:
	UF : 0, UT : 6,		CONFIG : 'N U T, 0, 0, 0',
	X =  230.672  mm,	Y =   -647.443  mm,	Z =   -248.118  mm,
	W =  90.000 deg,	P =   0.000 deg,	R =   90.000 deg
};
P[640]{
   GP1:
	UF : 0, UT : 6,		CONFIG : 'N U T, 0, 0, 0',
	X =  212.317  mm,	Y =   -657.957  mm,	Z =   -248.322  mm,
	W =  90.000 deg,	P =   0.000 deg,	R =   90.000 deg
};
P[641]{
   GP1:
	UF : 0, UT : 6,		CONFIG : 'N U T, 0, 0, 0',
	X =  194.250  mm,	Y =   -668.513  mm,	Z =   -248.021  mm,
	W =  90.000 deg,	P =   0.000 deg,	R =   90.000 deg
};
P[642]{
   GP1:
	UF : 0, UT : 6,		CONFIG : 'N U T, 0, 0, 0',
	X =  176.040  mm,	Y =   -679.034  mm,	Z =   -248.005  mm,
	W =  90.000 deg,	P =   0.000 deg,	R =   90.000 deg
};
P[643]{
   GP1:
	UF : 0, UT : 6,		CONFIG : 'N U T, 0, 0, 0',
	X =  157.868  mm,	Y =   -689.424  mm,	Z =   -248.251  mm,
	W =  90.000 deg,	P =   0.000 deg,	R =   90.000 deg
};
/END
